(* IEC 61131-3 sources: mect_apps/TP1043_RTU/Wattmeter_PLC, 6 files *)

(* ---- Crosstable.gvl ---- *)
VAR_GLOBAL
Potenza AT %QW0.772:UINT;
Tensione AT %QW0.776:UINT;
Potenza_Critica AT %IX0.780.0:BOOL;
Potenza_Distacco AT %IX0.784.0:BOOL;
V_L1_N AT %IW0.804:UINT;
A_L1 AT %IW0.808:UINT;
W_L1 AT %IW0.812:UINT;
VT_RATIO AT %IW0.840:UINT;
CT_RATIO AT %IW0.844:UINT;
RTU0_TYPE_PORT AT %ID0.20000:UDINT;
RTU0_BAUDRATE AT %ID0.20004:UDINT;
RTU0_STATUS AT %ID0.20008:UDINT;
RTU0_READS AT %ID0.20012:UDINT;
RTU0_WRITES AT %ID0.20016:UDINT;
RTU0_TIMEOUTS AT %ID0.20020:UDINT;
RTU0_COMM_ERRORS AT %ID0.20024:UDINT;
RTU0_LAST_ERROR AT %ID0.20028:UDINT;
RTU0_WRITE_QUEUE AT %ID0.20032:UDINT;
RTU0_READ_QUEUE AT %ID0.20036:UDINT;
TCPS_TYPE_PORT AT %ID0.20200:UDINT;
TCPS_IP_ADDRESS AT %ID0.20204:UDINT;
TCPS_STATUS AT %ID0.20208:UDINT;
TCPS_READS AT %ID0.20212:UDINT;
TCPS_WRITES AT %ID0.20216:UDINT;
TCPS_TIMEOUTS AT %ID0.20220:UDINT;
TCPS_COMM_ERRORS AT %ID0.20224:UDINT;
TCPS_LAST_ERROR AT %ID0.20228:UDINT;
TCPS_WRITE_QUEUE AT %ID0.20232:UDINT;
TCPS_READ_QUEUE AT %ID0.20236:UDINT;
NODE_01_DEV_NODE AT %ID0.20688:UDINT;
NODE_01_STATUS AT %ID0.20692:UDINT;
NODE_02_DEV_NODE AT %ID0.20696:UDINT;
NODE_02_STATUS AT %ID0.20700:UDINT;
NODE_03_DEV_NODE AT %ID0.20704:UDINT;
NODE_03_STATUS AT %ID0.20708:UDINT;
PLC_time AT %ID0.21560:REAL;
PLC_timeMin AT %ID0.21564:REAL;
PLC_timeMax AT %ID0.21568:REAL;
PLC_timeWin AT %QD0.21572:REAL;
PLC_Version AT %IW0.21576:UINT;
PLC_EngineStatus AT %IW0.21580:UINT;
PLC_ResetValues AT %QX0.21584.0:BOOL;
END_VAR

(* ---- Alarms.st ---- *)
(*[[
]]*)
PROGRAM Alarms
#import "Crosstable.gvl"
#import "Resource1.gvl"
VAR
END_VAR

;
END_PROGRAM

(* ---- Events.st ---- *)
(*[[
]]*)
PROGRAM Events
#import "Crosstable.gvl"
#import "Resource1.gvl"
VAR
END_VAR

;
END_PROGRAM

(* ---- Fast.st ---- *)
(*[[
]]*)
PROGRAM Fast
#import "Crosstable.gvl"
#import "Resource1.gvl"
VAR
END_VAR

;
END_PROGRAM

(* ---- Normal.st ---- *)
(*[[
]]*)
PROGRAM Normal
#import "Crosstable.gvl"
#import "Resource1.gvl"
VAR
	current_ratio : int;
END_VAR;

	current_ratio := CT_RATIO;
	if current_ratio = 0 then
		current_ratio := 4;
	end_if;

	Potenza := W_L1 * (VT_RATIO / 10) * current_ratio; (* P 111.1 *)
	Tensione := V_L1_N * (VT_RATIO / 10); (* VN 111.1 *)

END_PROGRAM

(* ---- Program1.st ---- *)
(*[[
]]*)
PROGRAM Program1

#import "Crosstable.gvl"
VAR
	current_ratio : int;
	first : bool := true;
END_VAR;
	if first then
		first := false;
		PLC_timeWin := 60.0;
	end_if;
	current_ratio := CT_RATIO;
	if current_ratio = 0 then
		current_ratio := 4;
	end_if;
	Potenza := W_L1 * (VT_RATIO / 10) * current_ratio; (* P 111.1 *)
	Tensione := V_L1_N * (VT_RATIO / 10); (* VN 111.1 *)

END_PROGRAM
